FUNCTION_BLOCK ""
{ S7_Optimized_Access := 'TRUE' }


END_FUNCTION_BLOCK
